TYPE "ProjectInfo"
VERSION : 0.1
// Block: ProjectInfo
   STRUCT
      Job : "String[20]";
      Revision : "String[10]";
      RevisionDate : DTL;
      Programmer : "String[20]";
      F_Signature : DWord;
      F_CompilationDate : DTL;
   END_STRUCT;

END_TYPE
